Yaskawa INFORM job: mataf_small_cylinder_program.JBI

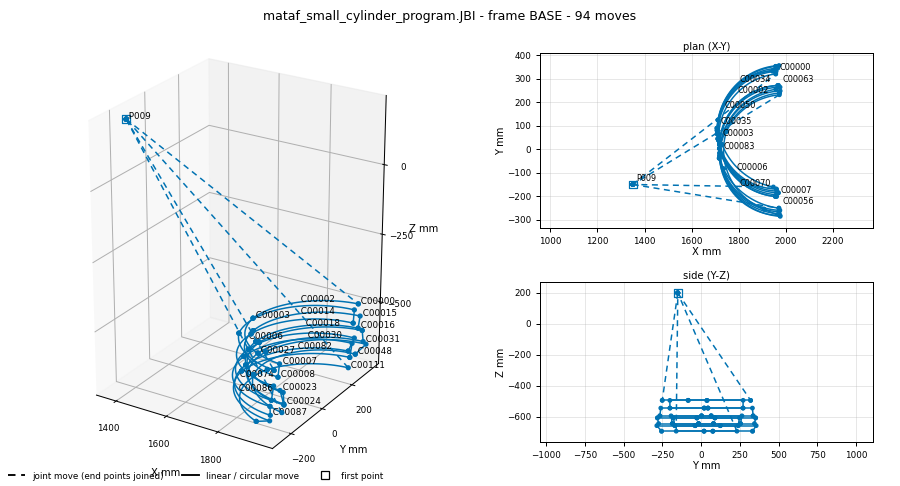
[picture p0: tool path of mataf_small_cylinder_program.JBI in frame BASE, 94 of 122 moves have a stored position in this frame; points joined in program order, loops and branches not executed]
/JOB
//NAME mataf_small_cylinder_program
//POS
///NPOS 112,0,112,1,0,4
///TOOL 0
///POSTYPE BASE
///RECTAN
///RCONF 0,0,0,0,0,0,0,0,0,0,0,0,0,0,0,0,0,0,0,0,0,0,0,0
C00000=1957.478,319.852,-493.161,93.3371,-90.0000,5.0000
C00001=1957.478,319.852,-493.161,93.3371,-90.0000,5.0000
C00002=1777.811,221.955,-493.161,142.9890,-90.0000,5.0000
C00003=1714.501,38.130,-493.161,-171.6714,-90.0000,5.0000
C00004=1714.501,38.130,-493.161,-171.6714,-90.0000,5.0000
C00005=1714.501,38.130,-493.161,-171.6714,-90.0000,5.0000
C00006=1773.821,-104.660,-493.161,-137.6397,-89.9999,5.0000
C00007=1961.271,-201.221,-493.161,-92.1580,-90.0000,5.0000
C00008=1955.524,-200.712,-542.798,-93.3502,-89.9999,5.0000
C00009=1955.524,-200.712,-542.798,-93.3502,-89.9999,5.0000
C00010=1792.548,-126.436,-542.798,-131.5398,-89.9999,5.0000
C00011=1711.565,44.458,-542.798,-173.1336,-89.9999,5.0000
C00012=1711.565,44.458,-542.798,-173.1336,-89.9999,5.0000
C00013=1711.565,44.458,-542.798,-173.1336,-89.9999,5.0000
C00014=1772.683,234.532,-542.798,141.4233,-89.9999,5.0000
C00015=1959.306,331.273,-542.798,92.7794,-90.0000,5.0000
C00016=1949.898,335.950,-592.798,94.7923,-90.0000,5.0000
C00017=1949.898,335.950,-592.798,94.7923,-90.0000,5.0000
C00018=1783.768,252.836,-592.798,136.7088,-90.0000,5.0000
C00019=1708.911,65.187,-592.798,-177.6909,-90.0000,5.0000
C00020=1708.911,65.187,-592.798,-177.6909,-90.0000,5.0000
C00021=1708.911,65.187,-592.798,-177.6909,-90.0000,5.0000
C00022=1791.202,-118.042,-592.798,-132.9621,-90.0000,5.0000
C00023=1959.265,-193.501,-592.798,-92.6459,-89.9999,5.0000
C00024=1968.704,-185.475,-642.798,-90.6590,-89.9999,5.0000
C00025=1968.704,-185.475,-642.798,-90.6590,-89.9999,5.0000
C00026=1789.487,-109.485,-642.798,-134.5249,-90.0000,5.0000
C00027=1708.391,80.274,-642.798,179.0231,-90.0000,5.0000
C00028=1708.391,80.274,-642.798,179.0231,-90.0000,5.0000
C00029=1708.391,80.274,-642.798,179.0231,-90.0000,5.0000
C00030=1785.471,261.068,-642.798,135.1471,-90.0000,5.0000
C00031=1966.164,344.443,-642.798,91.1825,-89.9999,5.0000
C00032=1957.256,352.172,-606.195,-180.0000,-60.0000,-87.0065
C00033=1957.256,352.172,-606.195,-180.0000,-60.0000,-87.0065
C00034=1789.254,270.033,-606.195,180.0000,-60.0000,-46.7932
C00035=1708.039,89.402,-606.195,180.0000,-60.0000,-2.9565
C00036=1708.039,89.402,-606.195,180.0000,-60.0000,-2.9565
C00037=1708.039,89.402,-606.195,180.0000,-60.0000,-2.9565
C00038=1781.217,-96.248,-606.195,180.0000,-60.0000,42.0849
C00039=1962.012,-178.006,-606.195,180.0000,-60.0000,87.8118
C00040=1960.296,-169.455,-656.195,180.0000,-60.0000,87.3353
C00041=1960.296,-169.455,-656.195,180.0000,-60.0000,87.3353
C00042=1763.513,-69.910,-656.195,180.0000,-60.0000,34.9841
C00043=1712.083,124.016,-656.195,180.0000,-60.0000,-10.5241
C00044=1712.083,124.016,-656.195,180.0000,-60.0000,-10.5241
C00045=1712.083,124.016,-656.195,180.0000,-60.0000,-10.5241
C00046=1806.529,290.057,-656.195,180.0000,-60.0000,-52.3718
C00047=1971.451,355.604,-656.195,180.0000,-60.0000,-89.9470
C00048=1943.582,332.180,-691.768,180.0000,-60.0000,-83.7395
C00049=1943.582,332.180,-691.768,180.0000,-60.0000,-83.7395
C00050=1724.057,160.346,-691.768,-180.0000,-60.0000,-18.8526
C00051=1729.523,19.353,-691.768,180.0000,-60.0000,13.1163
C00052=1729.523,19.353,-691.768,180.0000,-60.0000,13.1163
C00053=1729.523,19.353,-691.768,180.0000,-60.0000,13.1163
C00054=1821.468,-103.130,-691.768,180.0000,-60.0000,49.9785
C00055=1947.414,-160.456,-691.768,180.0000,-60.0000,84.1283
C00056=1970.823,-250.396,-492.768,-91.7483,-90.0000,5.0000
C00057=1970.823,-250.396,-492.768,-91.7483,-90.0000,5.0000
C00058=1845.933,-205.940,-492.768,-123.4754,-90.0000,5.0000
C00059=1734.867,-83.159,-492.768,-162.3665,-90.0000,5.0000
C00060=1734.867,-83.159,-492.768,-162.3665,-90.0000,5.0000
C00061=1734.867,-83.159,-492.768,-162.3665,-90.0000,5.0000
C00062=1727.760,81.156,-492.768,160.8616,-90.0000,5.0000
C00063=1969.335,271.334,-492.768,91.8506,-90.0000,5.0000
C00064=1966.184,270.952,-542.798,92.5046,-90.0000,5.0000
C00065=1966.184,270.952,-542.798,92.5046,-90.0000,5.0000
C00066=1797.296,196.487,-542.798,131.8221,-90.0000,5.0000
C00067=1718.146,20.262,-542.798,174.2822,-90.0000,5.0000
C00068=1718.146,20.262,-542.798,174.2822,-90.0000,5.0000
C00069=1718.146,20.262,-542.798,174.2822,-90.0000,5.0000
C00070=1786.351,-172.728,-542.798,-138.9840,-89.9999,5.0000
C00071=1975.114,-259.719,-542.798,-90.7165,-89.9999,5.0000
C00072=1970.775,-265.730,-592.798,-91.6557,-89.9999,5.0000
C00073=1970.775,-265.730,-592.798,-91.6557,-89.9999,5.0000
C00074=1790.943,-183.983,-592.798,-136.4333,-90.0000,5.0000
C00075=1717.978,3.173,-592.798,178.0291,-90.0000,5.0000
C00076=1717.978,3.173,-592.798,178.0291,-90.0000,5.0000
C00077=1717.978,3.173,-592.798,178.0291,-90.0000,5.0000
C00078=1790.048,182.261,-592.798,135.0297,-90.0000,5.0000
C00079=1975.876,263.645,-592.798,90.5132,-89.9999,5.0000
C00080=1958.655,254.696,-642.798,94.3107,-90.0000,5.0000
C00081=1958.655,254.696,-642.798,94.3107,-90.0000,5.0000
C00082=1798.690,173.735,-642.798,135.0126,-90.0000,5.0000
C00083=1719.649,-16.116,-642.798,-177.7124,-90.0000,5.0000
C00084=1719.649,-16.116,-642.798,-177.7124,-90.0000,5.0000
C00085=1719.649,-16.116,-642.798,-177.7124,-90.0000,5.0000
C00086=1790.601,-190.467,-642.798,-135.4624,-90.0000,5.0000
C00087=1972.001,-273.788,-642.798,-91.3442,-90.0000,5.0000
C00088=1975.087,-281.476,-606.195,-180.0000,-60.0000,89.3345
C00089=1975.087,-281.476,-606.195,-180.0000,-60.0000,89.3345
C00090=1789.810,-201.391,-606.195,180.0000,-60.0000,46.0631
C00091=1719.464,-27.068,-606.195,-180.0000,-60.0000,4.7010
C00092=1719.464,-27.068,-606.195,-180.0000,-60.0000,4.7010
C00093=1719.464,-27.068,-606.195,-180.0000,-60.0000,4.7010
C00094=1785.394,154.308,-606.195,180.0000,-60.0000,-39.6909
C00095=1976.406,247.905,-606.195,180.0000,-60.0000,-89.5745
C00096=1973.546,239.221,-656.195,180.0000,-60.0000,-88.8908
C00097=1973.546,239.221,-656.195,180.0000,-60.0000,-88.8908
C00098=1768.940,119.915,-656.195,180.0000,-60.0000,-30.9819
C00099=1717.413,-38.176,-656.195,180.0000,-60.0000,7.0779
C00100=1717.413,-38.176,-656.195,180.0000,-60.0000,7.0779
C00101=1717.413,-38.176,-656.195,180.0000,-60.0000,7.0779
C00102=1807.968,-213.750,-656.195,180.0000,-60.0000,50.6830
C00103=1976.542,-285.359,-656.195,180.0000,-60.0000,89.6418
C00104=1907.722,-254.667,-691.915,180.0000,-60.0000,74.1699
C00105=1907.722,-254.667,-691.915,180.0000,-60.0000,74.1699
C00106=1744.627,-71.845,-691.915,180.0000,-60.0000,15.7866
C00107=1748.184,76.066,-691.915,-180.0000,-60.0000,-19.5810
C00108=1748.184,76.066,-691.915,-180.0000,-60.0000,-19.5810
C00109=1748.184,76.066,-691.915,-180.0000,-60.0000,-19.5810
C00110=1836.206,180.579,-691.915,-180.0000,-60.0000,-52.6780
C00111=1973.009,231.266,-691.915,180.0000,-60.0000,-88.7238
///POSTYPE PULSE
///PULSE
EC00000=0
EC00001=0
EC00002=0
EC00003=0
EC00004=0
EC00005=0
EC00006=0
EC00007=0
EC00008=0
EC00009=0
EC00010=0
EC00011=0
EC00012=0
EC00013=0
EC00014=0
EC00015=0
EC00016=0
EC00017=0
EC00018=0
EC00019=0
EC00020=0
EC00021=0
EC00022=0
EC00023=0
EC00024=0
EC00025=0
EC00026=0
EC00027=0
EC00028=0
EC00029=0
EC00030=0
EC00031=0
EC00032=0
EC00033=0
EC00034=0
EC00035=0
EC00036=0
EC00037=0
EC00038=0
EC00039=0
EC00040=0
EC00041=0
EC00042=0
EC00043=0
EC00044=0
EC00045=0
EC00046=0
EC00047=0
EC00048=0
EC00049=0
EC00050=0
EC00051=0
EC00052=0
EC00053=0
EC00054=0
EC00055=0
EC00056=184320
EC00057=184320
EC00058=184320
EC00059=184320
EC00060=184320
EC00061=184320
EC00062=184320
EC00063=184320
EC00064=184320
EC00065=184320
EC00066=184320
EC00067=184320
EC00068=184320
EC00069=184320
EC00070=184320
EC00071=184320
EC00072=184320
EC00073=184320
EC00074=184320
EC00075=184320
EC00076=184320
EC00077=184320
EC00078=184320
EC00079=184320
EC00080=184320
EC00081=184320
EC00082=184320
EC00083=184320
EC00084=184320
EC00085=184320
EC00086=184320
EC00087=184320
EC00088=184320
EC00089=184320
EC00090=184320
EC00091=184320
EC00092=184320
EC00093=184320
EC00094=184320
EC00095=184320
EC00096=184320
EC00097=184320
EC00098=184320
EC00099=184320
EC00100=184320
EC00101=184320
EC00102=184320
EC00103=184320
EC00104=184320
EC00105=184320
EC00106=184320
EC00107=184320
EC00108=184320
EC00109=184320
EC00110=184320
EC00111=184320
///POSTYPE BASE
///RECTAN
///RCONF 1,0,0,0,0,0,0,0,0,0,0,0,0,0,0,0,0,0,0,0,0,0,0,0
P00009=1350.000,-150.000,200.000,-180.0000,-45.0000,0.0000
///POSTYPE PULSE
///PULSE
EX00000=92160
EX00001=184320
EX00002=276480
EX00003=368640
//INST
///DATE 2023/07/11 12:06
///ATTR SC,RW,RJ
////FRAME BASE
///GROUP1 RB1,ST1
NOP
MOVJ P009 EX000 VJ=15.00
MOVJ P009 VJ=15.00
MOVJ C00000 EC00000 VJ=15.00
CALL JOB:SPYON
MOVC C00001 EC00001 V=150.0
MOVC C00002 EC00002 V=150.0
MOVC C00003 EC00003 V=150.0
MOVL C00004 EC00004 V=150.0
MOVC C00005 EC00005 V=150.0
MOVC C00006 EC00006 V=150.0
MOVC C00007 EC00007 V=150.0
MOVL C00008 EC00008 V=150.0
MOVC C00009 EC00009 V=150.0
MOVC C00010 EC00010 V=150.0
MOVC C00011 EC00011 V=150.0
MOVL C00012 EC00012 V=150.0
MOVC C00013 EC00013 V=150.0
MOVC C00014 EC00014 V=150.0
MOVC C00015 EC00015 V=150.0
MOVL C00016 EC00016 V=150.0
MOVC C00017 EC00017 V=150.0
MOVC C00018 EC00018 V=150.0
MOVC C00019 EC00019 V=150.0
MOVL C00020 EC00020 V=150.0
MOVC C00021 EC00021 V=150.0
MOVC C00022 EC00022 V=150.0
MOVC C00023 EC00023 V=150.0
MOVL C00024 EC00024 V=150.0
MOVC C00025 EC00025 V=150.0
MOVC C00026 EC00026 V=150.0
MOVC C00027 EC00027 V=150.0
MOVL C00028 EC00028 V=150.0
MOVC C00029 EC00029 V=150.0
MOVC C00030 EC00030 V=150.0
MOVC C00031 EC00031 V=150.0
MOVL C00032 EC00032 V=150.0
MOVC C00033 EC00033 V=150.0
MOVC C00034 EC00034 V=150.0
MOVC C00035 EC00035 V=150.0
MOVL C00036 EC00036 V=150.0
MOVC C00037 EC00037 V=150.0
MOVC C00038 EC00038 V=150.0
MOVC C00039 EC00039 V=150.0
MOVL C00040 EC00040 V=150.0
MOVC C00041 EC00041 V=150.0
MOVC C00042 EC00042 V=150.0
MOVC C00043 EC00043 V=150.0
MOVL C00044 EC00044 V=150.0
MOVC C00045 EC00045 V=150.0
MOVC C00046 EC00046 V=150.0
MOVC C00047 EC00047 V=150.0
MOVL C00048 EC00048 V=150.0
MOVC C00049 EC00049 V=150.0
MOVC C00050 EC00050 V=150.0
MOVC C00051 EC00051 V=150.0
MOVL C00052 EC00052 V=150.0
MOVC C00053 EC00053 V=150.0
MOVC C00054 EC00054 V=150.0
MOVC C00055 EC00055 V=150.0
CALL JOB:SPYOF
MOVJ P009 VJ=15.00
MOVL P009 EX000 V=150.0
MOVJ P009 VJ=15.00
MOVL P009 EX001 V=150.0
MOVJ C00056 EC00056 VJ=15.00
CALL JOB:SPYON
MOVC C00057 EC00057 V=150.0
MOVC C00058 EC00058 V=150.0
MOVC C00059 EC00059 V=150.0
MOVL C00060 EC00060 V=150.0
MOVC C00061 EC00061 V=150.0
MOVC C00062 EC00062 V=150.0
MOVC C00063 EC00063 V=150.0
MOVL C00064 EC00064 V=150.0
MOVC C00065 EC00065 V=150.0
MOVC C00066 EC00066 V=150.0
MOVC C00067 EC00067 V=150.0
MOVL C00068 EC00068 V=150.0
MOVC C00069 EC00069 V=150.0
MOVC C00070 EC00070 V=150.0
MOVC C00071 EC00071 V=150.0
MOVL C00072 EC00072 V=150.0
MOVC C00073 EC00073 V=150.0
MOVC C00074 EC00074 V=150.0
MOVC C00075 EC00075 V=150.0
MOVL C00076 EC00076 V=150.0
MOVC C00077 EC00077 V=150.0
MOVC C00078 EC00078 V=150.0
MOVC C00079 EC00079 V=150.0
MOVL C00080 EC00080 V=150.0
MOVC C00081 EC00081 V=150.0
MOVC C00082 EC00082 V=150.0
MOVC C00083 EC00083 V=150.0
MOVL C00084 EC00084 V=150.0
MOVC C00085 EC00085 V=150.0
MOVC C00086 EC00086 V=150.0
MOVC C00087 EC00087 V=150.0
MOVL C00088 EC00088 V=150.0
MOVC C00089 EC00089 V=150.0
MOVC C00090 EC00090 V=150.0
MOVC C00091 EC00091 V=150.0
MOVL C00092 EC00092 V=150.0
MOVC C00093 EC00093 V=150.0
MOVC C00094 EC00094 V=150.0
MOVC C00095 EC00095 V=150.0
MOVL C00096 EC00096 V=150.0
MOVC C00097 EC00097 V=150.0
MOVC C00098 EC00098 V=150.0
MOVC C00099 EC00099 V=150.0
MOVL C00100 EC00100 V=150.0
MOVC C00101 EC00101 V=150.0
MOVC C00102 EC00102 V=150.0
MOVC C00103 EC00103 V=150.0
MOVL C00104 EC00104 V=150.0
MOVC C00105 EC00105 V=150.0
MOVC C00106 EC00106 V=150.0
MOVC C00107 EC00107 V=150.0
MOVL C00108 EC00108 V=150.0
MOVC C00109 EC00109 V=150.0
MOVC C00110 EC00110 V=150.0
MOVC C00111 EC00111 V=150.0
CALL JOB:SPYOF
MOVJ P009 VJ=15.00
MOVL P009 EX002 V=150.0
MOVJ P009 VJ=15.00
MOVL P009 EX003 V=150.0
END
